Staubli VAL3: resumeCycle.pgx

public program resumeCycle()
begin
  if cycleStatus:bPause
    // resume the cycle
    logMsg("[KERNEL] CYCLE: Restart the cycle")
    cycleStatus:bToPause=true
    watch(cycleStatus:bToPause==false,1)
  endIf
end
